// TwinCAT 3 PLC project BRS2_Logic
// ProgramVersion: 3.1.0.9
// libraries:
//   Tc2_Standard, * (Beckhoff Automation GmbH)
//   Tc2_System, * (Beckhoff Automation GmbH)
//   Tc3_Interfaces, * (Beckhoff Automation GmbH)
//   Tc3_Module, * (Beckhoff Automation GmbH)
// project tree:
//   / PlcTask.TcTTO
//   POUs/ MAIN.TcPOU
// real-time tasks:
//   TASK PlcTask: cycle T#4ms, priority 20, ADS port 350
// I/O:
//   DEVICE Device 1 (EtherCAT), AmsNetId 10.0.0.103.2.1
//     Term 7 (EK1101) [EK1101 EtherCAT Coupler (2A E-Bus, ID switch)]
//       Term 9 (EL3202-0010) [EL3202-0010 2Ch. Ana. Input PT100 (RTD), High Precision]
//       Term 8 (EL2124) [EL2124 4Ch. Dig. Output 5V, 20mA]
//       Term 10 (EL4102) [EL4102 2Ch. Ana. Output  0-10V, 16bit]
//       Term 11 (EL2624) [EL2624 4Ch. Relay Output, NO (125V AC / 30V DC)]
//       Term 14 (EL9011) [EL9011 End Terminal]
//   DEVICE Device 2 (EtherCAT) (disabled), AmsNetId 10.0.0.103.3.1
//     Box 1 (EP4174-0002) [EP4174-0002 4Ch. Ana. Output +/-10V, 0-10V, 0/4-20mA configurable]
//     Box 2 (EP4374-0002) [EP4374-0002 2Ch. Ana. Input +/-10V, 0-10V, 0/4-20mA configurable; 2Ch. Ana. Output +/-10V, 0-10V, 0/4-20mA configurable]
// variable links:
//   BRS2_Logic/BRS2_Logic Instance <-> Device 1 (EtherCAT)/Term 7 (EK1101)/Term 10 (EL4102)
//     PlcTask Outputs/MAIN.OUT1 <-> Channel 1/Output
//     PlcTask Outputs/MAIN.OUT2 <-> Channel 2/Output
//   BRS2_Logic/BRS2_Logic Instance <-> Device 1 (EtherCAT)/Term 7 (EK1101)/Term 11 (EL2624)
//     PlcTask Outputs/MAIN.RELAYL <-> Channel 1/Output
//     PlcTask Outputs/MAIN.RELAYR <-> Channel 2/Output

CONFIGURATION BRS2_Logic
    RESOURCE PLC ON TwinCAT3
        TASK PlcTask(INTERVAL := T#4ms, PRIORITY := 20);
        PROGRAM MAIN WITH PlcTask : MAIN;
    END_RESOURCE
END_CONFIGURATION

// ---- POUs/MAIN.TcPOU
PROGRAM MAIN
VAR
	IN1 AT %MD0: INT;
	IN2 AT %MD1: INT;

	RELAYL AT %QW1: BOOL;
	RELAYR AT %QW2: BOOL;
	
	OUT1 AT %QW3: INT;
	OUT2 AT %QW4: INT;
	
	L: INT;
END_VAR

RELAYL:=TRUE;
RELAYR:=TRUE;

OUT1:=IN1;
OUT2:=IN2;

END_PROGRAM
